(* IEC 61131-3 sources: repolevel_ST_code_completion/output/0127完整版本_带planner/repoeval_electronic_cam_motion/readful_result_before_fix, 4 files *)

(* ---- F_AxisStatusToString.st ---- *)
FUNCTION F_AxisStatusToString : STRING
VAR_INPUT
	fbReadStatus	:	MC_ReadStatus;		//轴状态读取功能块
END_VAR
IF NOT fbReadStatus.Enable THEN
	F_AxisStatusToString := 'InvalidStatus';
	RETURN;
END_IF

IF fbReadStatus.Done THEN
	F_AxisStatusToString := 'MotionCompleted';
	RETURN;
END_IF

IF fbReadStatus.MotionActive THEN
	F_AxisStatusToString := 'InMotion';
	RETURN;
END_IF

IF fbReadStatus.ErrorActive THEN
	F_AxisStatusToString := 'ErrorState';
	RETURN;
END_IF

IF fbReadStatus.StandStill THEN
	F_AxisStatusToString := 'StandStill';
	RETURN;
END_IF

F_AxisStatusToString := 'UnknownStatus';
RETURN;
END_FUNCTION

(* ---- FB_DualAxisPower.st ---- *)
FUNCTION_BLOCK FB_DualAxisPower
VAR_INPUT
	Axis1			:	AXIS_REF;			//轴1引用
	Axis2			:	AXIS_REF;			//轴2引用
	bPowerOn		:	BOOL;				//电源使能信号
END_VAR
VAR_OUTPUT
	bPowerDone		:	BOOL;				//两轴都准备就绪
	bAxis1Ready		:	BOOL;				//轴1准备就绪
	bAxis2Ready		:	BOOL;				//轴2准备就绪
	bError			:	BOOL;				//错误标志
END_VAR
VAR
	fbPower1		:	MC_Power;			//轴1电源控制
	fbPower2		:	MC_Power;			//轴2电源控制
	bAxis1Error		:	BOOL;				//轴1错误标志
	bAxis2Error		:	BOOL;				//轴2错误标志
END_VAR

IF NOT bPowerOn THEN
	bPowerDone := FALSE;
	bAxis1Ready := FALSE;
	bAxis2Ready := FALSE;
	bError := FALSE;
	RETURN;
END_IF

// 执行轴1电源控制
fbPower1(
	Axis := Axis1,
	Enable := TRUE,
	bDriveStart := bPowerOn,
	bRegulatorOn := bPowerOn
);
bAxis1Ready := fbPower1.Status = MC_POWER_STATUS_READY;
bAxis1Error := fbPower1.Error;

// 执行轴2电源控制
fbPower2(
	Axis := Axis2,
	Enable := TRUE,
	bDriveStart := bPowerOn,
	bRegulatorOn := bPowerOn
);
bAxis2Ready := fbPower2.Status = MC_POWER_STATUS_READY;
bAxis2Error := fbPower2.Error;

// 判断两轴是否都准备就绪
IF bAxis1Ready AND bAxis2Ready THEN
	bPowerDone := TRUE;
ELSE
	bPowerDone := FALSE;
END_IF

// 检测是否出现错误
IF bAxis1Error OR bAxis2Error THEN
	bError := TRUE;
ELSE
	bError := FALSE;
END_IF
END_FUNCTION_BLOCK

(* ---- FB_DualAxisReset.st ---- *)
FUNCTION_BLOCK FB_DualAxisReset
VAR_INPUT
	Axis1			:	AXIS_REF;			//轴1引用
	Axis2			:	AXIS_REF;			//轴2引用
	bExecute		:	BOOL;				//执行复位信号
END_VAR
VAR_OUTPUT
	bDone			:	BOOL;				//复位完成
	bBusy			:	BOOL;				//复位进行中
	bError			:	BOOL;				//错误标志
END_VAR
VAR
	fbReset1		:	MC_Reset;			//轴1复位
	fbReset2		:	MC_Reset;			//轴2复位
	fbReadStatus1	:	MC_ReadStatus;		//轴1状态读取
	fbReadStatus2	:	MC_ReadStatus;		//轴2状态读取
	bError1			:	BOOL;				//轴1错误标志
	bError2			:	BOOL;				//轴2错误标志
	nState			:	UDINT;				//状态机
	tTimeout		:	TIME := T#5s;		//超时时间
	tStartTime		:	TIME;				//开始时间
END_VAR

CASE nState OF
	0: (* 空闲状态 *)
		bDone := FALSE;
		bBusy := FALSE;
		bError := FALSE;

		IF bExecute THEN
			bBusy := TRUE;
			tStartTime := TIME(); (* 记录开始时间 *)
			nState := 10;
		END_IF;

	10: (* 检查轴状态 *)
		fbReadStatus1(Axis := Axis1);
		fbReadStatus2(Axis := Axis2);

		bError1 := NOT fbReadStatus1.Error AND NOT fbReadStatus1.Valid;
		bError2 := NOT fbReadStatus2.Error AND NOT fbReadStatus2.Valid;

		IF bError1 OR bError2 THEN
			bError := TRUE;
			bBusy := FALSE;
			nState := 0;
		ELSE
			nState := 20;
		END_IF;

	20: (* 执行复位 *)
		fbReset1(Axis := Axis1, Execute := TRUE);
		fbReset2(Axis := Axis2, Execute := TRUE);

		IF fbReset1.Done AND fbReset2.Done THEN
			bDone := TRUE;
			bBusy := FALSE;
			bError := FALSE;
			nState := 0;
		ELSIF fbReset1.Error OR fbReset2.Error THEN
			bError := TRUE;
			bBusy := FALSE;
			bDone := FALSE;
			nState := 0;
		ELSIF (TIME() - tStartTime) > tTimeout THEN
			bError := TRUE;
			bBusy := FALSE;
			bDone := FALSE;
			nState := 0;
		END_IF;
END_CASE;
END_FUNCTION_BLOCK

(* ---- ResetAxis.st ---- *)
FUNCTION_BLOCK ResetAxis
VAR_INPUT
	bExec	:	BOOL;
END_VAR
VAR
	fbReset1	:	MC_Reset;
	fbReset2	:	MC_Reset;

	fbReadAxisError1	:	MC_ReadAxisError;
	fbReadAxisError2	:	MC_ReadAxisError;

	fbReadStatus1	:	MC_ReadStatus;
	fbReadStatus2	:	MC_ReadStatus;

	fbExecTrig	:	R_TRIG;
	nState 		:	BYTE;

	bErrorX		:	BOOL;
	bErrorY		:	BOOL;

	bResetDoneX	:	BOOL;
	bResetDoneY	:	BOOL;
END_VAR

VAR_OUTPUT
	Done	:	BOOL;
END_VAR

fbExecTrig(CLK := bExec);

CASE nState OF
	0:
		IF fbExecTrig.Q THEN
			nState := 1;
			Done := FALSE;
		END_IF

	1:
		fbReadAxisError1(Execute := TRUE);
		fbReadAxisError2(Execute := TRUE);
		bErrorX := fbReadAxisError1.ErrorID <> 0;
		bErrorY := fbReadAxisError2.ErrorID <> 0;

		IF NOT bErrorX AND NOT bErrorY THEN
			nState := 4;
		ELSE
			nState := 2;
		END_IF

	2:
		fbReset1(Execute := bErrorX);
		fbReset2(Execute := bErrorY);
		bResetDoneX := fbReset1.Done;
		bResetDoneY := fbReset2.Done;

		IF bResetDoneX OR bResetDoneY THEN
			nState := 3;
		END_IF

	3:
		fbReadStatus1(Enable := TRUE);
		fbReadStatus2(Enable := TRUE);

		IF fbReadStatus1.Error OR fbReadStatus2.Error THEN
			nState := 2;
		ELSIF fbReadStatus1.Valid AND fbReadStatus2.Valid THEN
			nState := 4;
		END_IF

	4:
		Done := TRUE;
		nState := 0;
END_CASE
END_FUNCTION_BLOCK
